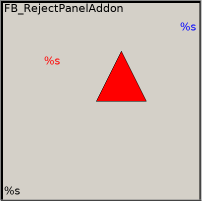
VISUALIZATION V_RejectPanelAddon  // 202x201
VAR_IN_OUT
	{attribute 'VAR_IN_OUT_AS_POINTER'}
	fbFunction		: FB_RejectPanelAddon;	
END_VAR
    Rectangle (1,1 200x200)
    Label (1,1 200x15), "FB_RejectPanelAddon"
    Rectangle (1,181 200x20), "%s", text variable: fbFunction.ConfigFunction.FunctionName
    Rectangle (41,51 161x20), "%s", text variable: fbFunction.ZoneData[1].ErrorData.Error.ErrorCode.Conv, invisible if: fbFunction.FunctionData.ErrorData.Error.ErrorCode.Conv = 0
    Polygon (96,101) (121,51) (146,101) (131,101) (111,101), invisible if: fbFunction.FunctionData.ErrorData.ErrorState = E_ErrorState.OPERATIONAL
    Rectangle (38,17 161x20), "%s", text variable: fbFunction.RejectPanelState.eState
END_VISUALIZATION

(* stored: Version 1.1.0.1, ProductVersion 3.1.4024.4
   Visu V_RejectPanelAddon: Id {b8ebb3bf-2612-4793-a502-d788b280e6e0} *)
